// TIA Portal V16 export
// export: Created 2022-04-14T22:38:50.7764666Z, ExportSetting WithDefaults, DisplayName Totally Integrated Automation Portal, DisplayVersion V16, DisplayName TIA Portal Version Control Interface, DisplayVersion V16, DisplayName TIA Portal Openness, DisplayVersion V16, DisplayName STEP 7 Professional, DisplayVersion V16, DisplayName STEP 7 Safety, DisplayVersion V16, DisplayName WinCC Professional, DisplayVersion V16
FUNCTION_BLOCK "Entry Conveyor"   // FB5, LAD
{ S7_Optimized_Access := 'TRUE' }
VERSION : 0.1
// stored: AutoNumber true, IsIECCheckEnabled false, IsRetainMemResEnabled false, MemoryReserve 100, SetENOAutomatically false, UDAEnableTagReadback false
BEGIN

REGION Network 1
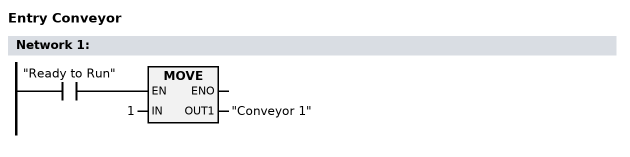
   RUNG wire#powerrail
      Contact( "Ready to Run" )
      Move(in := 1, out1 => "Conveyor 1")
   END_RUNG
   // the same network as SCL:
   IF "Ready to Run" THEN "Conveyor 1" := 1; END_IF;
END_REGION
END_FUNCTION_BLOCK
